SYSTEM Kulbana System 2
  (* Version 1.0, 2007-08-23, Goran, Chalmers *)
  DEVICE Test Device : DeviceType_not_used
    RESOURCE TestResource : ResourceType_not_used
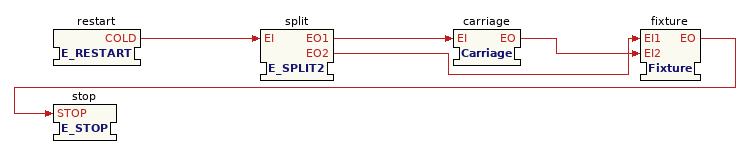
      FBS
        restart : E_RESTART;
        stop : E_STOP;
        split : E_SPLIT2;
        carriage : Carriage;
        fixture : Fixture;
      END_FBS
      EVENT_CONNECTIONS
        restart.COLD TO split.EI;
        split.EO1 TO carriage.EI;
        split.EO2 TO fixture.EI1;
        carriage.EO TO fixture.EI2;
        fixture.EO TO stop.STOP;
      END_CONNECTIONS
    END_RESOURCE
  END_DEVICE
END_SYSTEM
